# EPICS substitutions: es2-psu/es2-psu1.substitutions
file /epics/iocs/SorensonXG850/db/sorensonxg850-232.template
{
	pattern { Sys		, Dev		, PORT		, ADR	}
		{ XF:23ID2-ES	, "{PSU:1}"	, XF23ID2_PSU1	, 1	}
}
